VAR_GLOBAL
	HeatCurve	:	ARRAY[0..40,0..1] OF REAL;
END_VAR

(* stored: Version 1.1.0.1, ProductVersion 3.1.4018.2
   GVL HeatingCurve: Id {f585fd7d-37c8-4e56-a844-a3dfcb75af1e} *)
